/// Due to an increase in the use of solid-state sensors like proximity switches, this pattern will be less likely to be seen 
FUNCTION_BLOCK FbDebounce
VAR_INPUT
	xInput: BOOL;
END_VAR
VAR_OUTPUT
	xDebouncedInput: BOOL;
END_VAR
VAR
	DelayOn: Ton;
	tETon: TIME;
	DelayOff: Ton;
	tEToff: TIME;
END_VAR

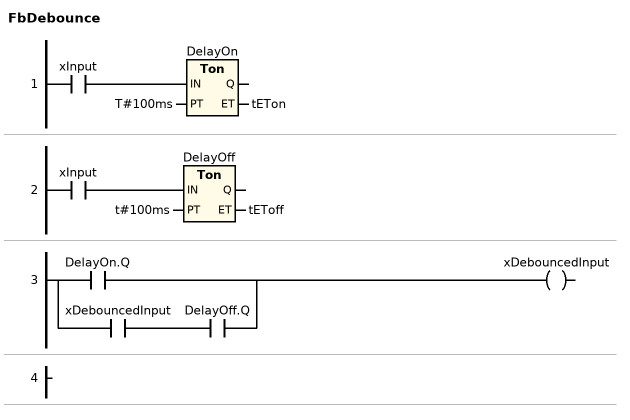
// NETWORK 1
DelayOn(IN := xInput, PT := T#100ms, ET => tETon); // Ton

// NETWORK 2
DelayOff(IN := xInput, PT := t#100ms, ET => tEToff); // Ton

// NETWORK 3
xDebouncedInput := DelayOn.Q OR xDebouncedInput AND DelayOff.Q;

// NETWORK 4

END_FUNCTION_BLOCK

(* stored: Version 1.1.0.1, ProductVersion 3.1.4024.12
   POU FbDebounce: Id {f3d9dc7e-70c3-4481-b21c-a508acbd7e24}, SpecialFunc None *)
